(* IEC 61131-3 sources: programs/VI-54/VI-54_20171205/VI-54_20171205/Stations/PLC_VI54/VI-54_171014/Class/ReleaseBrake, 1 file *)

(* ---- ReleaseBrake.st ---- *)
(*!
<Class
	Name               = "ReleaseBrake"
	Revision           = "0.1"
	RealtimeTask       = "false"
	CyclicTask         = "false"
	BackgroundTask     = "true"
	DefBackground      = "100 ms"
	Sigmatek           = "false"
	OSInterface        = "false"
	HighPriority       = "false"
	Automatic          = "false"
	UpdateMode         = "Prescan"
	SharedCommandTable = "true"
	Objectsize         = "(630,240)">
	<Channels>
		<Server Name="ActPosM1" Visualized="true" Initialize="false" WriteProtected="true" Retentive="false"/>
		<Server Name="Comm" Visualized="true" Initialize="false" WriteProtected="false" Retentive="false"/>
		<Client Name="_DriveParaBaseM1" Required="true" Internal="true"/>
		<Client Name="Axle" Required="true" Internal="false"/>
		<Client Name="iBrakeSwitch" Required="false" Internal="false"/>
		<Client Name="oReleaseBrake" Required="false" Internal="false"/>
	</Channels>
	<Network Name="ReleaseBrake">
		<!-- List of Components in this network -->
		<Components>
			<Object
				Name       = "_DriveParaBaseM1"
				Class      = "_DriveParaBase"
				Position   = "(330,120)"
				Visualized = "true">
				<Channels>
					<Server Name="State"/>
					<Client Name="DriveAxis"/>
					<Client Name="ErrorCode"/>
				</Channels>
			</Object>
		</Components>
		<Comments>
		</Comments>
		<!-- List of Connections in this network -->
		<Connections>
			<Connection Source="this._DriveParaBaseM1" Destination="_DriveParaBaseM1.State"/>
			<Connection Source="_DriveParaBaseM1.DriveAxis" Destination="this.Axle" Vertices="(330,210),(38,210),"/>
		</Connections>
		<!-- Headerfiles -->
		<Options>
		</Options>
	</Network>
</Class>
*)
ReleaseBrake : CLASS
  //Servers:
	Comm 	: SvrChCmd_DINT;
	ActPosM1 	: SvrCh_DINT;
  //Clients:
	Axle 	: CltChCmd__DriveAxis;
	iBrakeSwitch 	: CltCh_DINT;
	_DriveParaBaseM1 	: CltChCmd__DriveParaBase;
	oReleaseBrake 	: CltCh_DINT;
  //Variables:
		BrakeSwitchOld 	: DINT;
  //Functions:

	FUNCTION VIRTUAL GLOBAL Background
		VAR_INPUT
			EAX 	: UDINT;
		END_VAR
		VAR_OUTPUT
			state (EAX) 	: UDINT;
		END_VAR;

	FUNCTION GLOBAL NoBrake;
  //Tables:
	FUNCTION @STD
		VAR_OUTPUT
			ret_code	: CONFSTATES;
		END_VAR;
	FUNCTION GLOBAL TAB @CT_;
END_CLASS;

#pragma using _DriveParaBase
#pragma usingLtd _DriveAxis

FUNCTION VIRTUAL GLOBAL ReleaseBrake::Background
	VAR_INPUT
		EAX 	: UDINT;
	END_VAR
	VAR_OUTPUT
		state (EAX) 	: UDINT;
	END_VAR

  // brake control
  if Axle.AxEnable = 1 then
    iBrakeSwitch := 0;
    Comm := 0;
  else
    // Release brake
    if IsClientConnected(#iBrakeSwitch) then
      iBrakeSwitch := (iBrakeSwitch.Read() = 1 | Comm = 1);
    else
      iBrakeSwitch := Comm;
    end_if;
  end_if;

  ActPosM1 := Axle.ActPos;

// Release brake
  if ops.tAbsolute > 10000 then
    oReleaseBrake := 1;
    if IsClientConnected(#oReleaseBrake) then
      oReleaseBrake.Write (oReleaseBrake);
    end_if;
    if iBrakeSwitch <> BrakeSwitchOld then
      BrakeSwitchOld := iBrakeSwitch;
      _DriveParaBaseM1.SetASyncCmd(ParaNr:=222, ParaRdWr:=1, ParaValue := iBrakeSwitch, pThis:=this);
    end_if;
  end_if;

	state := READY;

END_FUNCTION

FUNCTION GLOBAL ReleaseBrake::NoBrake

  // When we use no brake
  _DriveParaBaseM1.SetASyncCmd(ParaNr:= SDD_M_BRAKE, ParaRdWr:= 1, ParaValue:= 0, pThis:= this);

END_FUNCTION
